// TwinCAT 3 PLC project LEO_Demo
// ProgramVersion: 3.1.4023.0
// libraries:
//   EfficientIO Communicator, * (EfficientIO)
//   Tc2_BABasic, * (Beckhoff Automation GmbH)
//   Tc2_Standard, * (Beckhoff Automation GmbH)
//   Tc2_System, * (Beckhoff Automation GmbH)
//   Tc2_Utilities, * (Beckhoff Automation GmbH)
//   Tc3_Module, * (Beckhoff Automation GmbH)
// project tree:
//   / FastTask.TcTTO, PlcTask.TcTTO, SlowTask.TcTTO
//   GVLs/ GVL.TcGVL
//   POUs/ prgComLynus.TcPOU, prgCS.TcPOU, prgEM.TcPOU, prgGrid.TcPOU, prgLightSwitch.TcPOU, prgPV.TcPOU, prgReadWrite.TcPOU, prgSun.TcPOU, prgSystemTime.TcPOU, prgVarInfo.TcPOU
// real-time tasks:
//   TASK MiddleTask: cycle T#10ms, priority 8, ADS port 350
//   TASK SlowTask: cycle T#20ms, priority 10, ADS port 351
//   TASK FastTask: cycle T#5ms, priority 6, ADS port 352

CONFIGURATION LEO_Demo
    RESOURCE PLC ON TwinCAT3
        TASK FastTask(INTERVAL := T#5ms, PRIORITY := 6);
        TASK PlcTask(INTERVAL := T#10ms, PRIORITY := 8);
        TASK SlowTask(INTERVAL := T#20ms, PRIORITY := 10);
        PROGRAM prgVarInfo WITH FastTask : prgVarInfo;
        PROGRAM prgReadWrite WITH FastTask : prgReadWrite;
        PROGRAM prgEM WITH PlcTask : prgEM;
        PROGRAM prgLightSwitch WITH PlcTask : prgLightSwitch;
        PROGRAM prgCS WITH PlcTask : prgCS;
        PROGRAM prgPV WITH PlcTask : prgPV;
        PROGRAM prgGrid WITH PlcTask : prgGrid;
        PROGRAM prgSystemTime WITH PlcTask : prgSystemTime;
        PROGRAM prgSun WITH PlcTask : prgSun;
        PROGRAM prgComLynus WITH SlowTask : prgComLynus;
    END_RESOURCE
END_CONFIGURATION

// ---- GVLs/GVL.TcGVL
{attribute 'qualified_only'}
VAR_GLOBAL
	location_lat	: LREAL; //{#lynus.ag#()}
	location_lon	: LREAL; //{#lynus.ag#()}
END_VAR

// ---- POUs/prgVarInfo.TcPOU
PROGRAM prgVarInfo
VAR
	fbVar			: FB_VarInfo;
END_VAR

fbVar(
	bReadInfo:= , 
	eTMCFile:= eSelectTMCFile.eDontUseTMCFile, 
	eSavePositionTMCFile:= eSavePositionOnPLC.ePostionC, 
	udiCounterFoundVariables=> , 
	bError=> , 
	bBusy=> , 
	byProgress=> , 
	udiErrorCodeOut=> , 
	eErrorVarInfo_Out=> , 
	sVarWithError=> );

END_PROGRAM

// ---- POUs/prgReadWrite.TcPOU
PROGRAM prgReadWrite
VAR
	fbRW		: FB_ReadWrite;
END_VAR

fbRW(bBusy=> , bError=> , udiErrorCodeOut=> , eErrorReadWrite_Out=> );

END_PROGRAM

// ---- POUs/prgEM.TcPOU
PROGRAM prgEM
VAR
	fbRand			: DRAND;
	lrRandNum		: LREAL;
	lrEMConsumption	: LREAL; //{#lynus.ag#()}
	lrEMCounter		: LREAL; //{#lynus.ag#()}
	fbTimer1		: TON;
	bStart1			: BOOL := TRUE;
	fbTimer2		: TON;
	bStart2			: BOOL;
END_VAR

fbTimer1(IN := bStart1, PT := T#15M);

IF fbTimer1.Q THEN
	bStart1 := FALSE;
	fbRand(Seed := 0);
	lrEMConsumption := fbRand.Num / 2;
	lrEMCounter := lrEMCounter + lrEMConsumption;
	bStart2 := TRUE;
END_IF

fbTimer2(IN := bStart2, PT := T#15M);

IF fbTimer2.Q THEN
	bStart2 := FALSE;
	fbRand(Seed := 0);
	lrEMConsumption := fbRand.Num;
	bStart1 := TRUE;
	lrEMCounter := lrEMCounter + lrEMConsumption;
END_IF

END_PROGRAM

// ---- POUs/prgLightSwitch.TcPOU
PROGRAM prgLightSwitch
VAR
	fbLight : FB_Light;
	bSwitchOn : BOOL; //{#lynus.ag#()}
	bSwitchOff : BOOL; //{#lynus.ag#()}
	bStateLight : BOOL; //{#lynus.ag#()}
END_VAR

fbLight(bOn:=bSwitchOn, bOff:=bSwitchOff, bLight=>bStateLight);

END_PROGRAM

// ---- POUs/prgCS.TcPOU
PROGRAM prgCS
VAR
	fbCSvirt	: FB_Light;
	bCSOn		: BOOL; //{#lynus.ag#()}
	bCSOff		: BOOL; //{#lynus.ag#()}
	bStateCS	: BOOL; //{#lynus.ag#()}
	lrCSpower	: LREAL; //{#lynus.ag#()}
END_VAR

fbCSvirt(bOn:=bCSOn, bOff:=bCSOff, bLight=>bStateCS);

IF bStateCS THEN
	lrCSpower := 11.02;
	ELSE
	lrCSpower := 0;
END_IF

END_PROGRAM

// ---- POUs/prgPV.TcPOU
PROGRAM prgPV
VAR
	fbPVvirt	: FB_Light;
	bPVOn		: BOOL; //{#lynus.ag#()}
	bPVOff		: BOOL; //{#lynus.ag#()}
	bStatePV	: BOOL; //{#lynus.ag#()}
	lrPVpower	: LREAL; //{#lynus.ag#()}
END_VAR

fbPVvirt(bOn:=bPVOn, bOff:=bPVOff, bLight=>bStatePV);

IF bStatePV THEN
	lrPVpower := 9.72;
	ELSE
	lrPVpower := 0;
END_IF

END_PROGRAM

// ---- POUs/prgGrid.TcPOU
PROGRAM prgGrid
VAR
	lrGridPower	: LREAL; //{#lynus.ag#()}
END_VAR

lrGridPower := prgEM.lrEMConsumption + prgCS.lrCSpower - prgPV.lrPVpower;

END_PROGRAM

// ---- POUs/prgSystemTime.TcPOU
PROGRAM prgSystemTime
VAR
	fbGetTime			: NT_GetTime;
	dtSystemTime		: DT;
	stDateTime			: TIMESTRUCT;
	tonGetTime			: TON;
	nStep				: INT;
	bSystemTimeValid	: BOOL := FALSE;
END_VAR

CASE nStep OF
0:
	tonGetTime(IN:=TRUE, PT:=T#500MS);
	IF (tonGetTime.Q) THEN
		tonGetTime(IN := FALSE);
		nStep:=10;
	END_IF

10:
	fbGetTime(NETID:='', START:=TRUE, TMOUT:=T#2S);
	IF (NOT fbGetTime.BUSY) THEN
		stDateTime := fbGetTime.TIMESTR;
		dtSystemTime := SYSTEMtimE_TO_DT(fbGetTime.TIMESTR);
		fbGetTime(START := FALSE);
		bSystemTimeValid := TRUE;
		nStep := 0;
	END_IF	
END_CASE

END_PROGRAM

// ---- POUs/prgSun.TcPOU
PROGRAM prgSun
VAR
	fbTimerC1					: FB_WeeklyTimeSwitch;
	fbCalcSunriseSunset   		: FB_CalcSunriseSunset;
	todSunrise            		: TOD;
	todSunset             		: TOD;
	bCircle1On					: BOOL;
	bCircle1Off					: BOOL;
	tSwitchOnTime				: TOD;	//{#lynus.ag#()}
	tSwitchOffTime				: TOD;	//{#lynus.ag#()}
END_VAR

VAR PERSISTENT
	bEnableTimerC1				: BOOL;
END_VAR


IF prgSystemTime.bSystemTimeValid THEN

	fbCalcSunriseSunset(
		fDegreeOfLongitude := GVL.location_lon,   (* Longitude of Verl *)
        fDegreeOfLatitude := GVL.location_lat,   (* Latitude of Verl *)
    	fReferenceMeridian := 30.0,  (* Central European Summer Time *)
        dCurrentDate := DT_TO_DATE(prgSystemTime.dtSystemTime),
        todSunrise => todSunrise,
        todSunset => todSunset);
END_IF


(*
IF prgSystemTime.bSystemTimeValid THEN

	fbTimerC1(
		bEnable:=bEnableTimerC1, 
		tCurrentDateTime:=prgSystemTime.dtSystemTime, 
		tSwitchOnTime:=todSunrise, 
		tSwitchOffTime:=todSunset, 
		bSunday:=TRUE, 
		bMonday:=TRUE, 
		bTuesday:=TRUE, 
		bWednesday:=TRUE, 
		bThursday:=TRUE, 
		bFriday:=TRUE, 
		bSaturday:=TRUE,
		bEdgeOn=> bCircle1On,
		bEdgeOff=> bCircle1Off);
END_IF
*)

END_PROGRAM

// ---- POUs/prgComLynus.TcPOU
PROGRAM prgComLynus
VAR
	fbCom			: FB_MqttCommunicator;
END_VAR

fbCom(
	bConnect:= TRUE, 
	sUserName:= 'c43048fc-b368-4152-a20e-2efdedf6f25a', 
	sUserPassword:= 'a3dbe556-ed89-450d-a0be-4c95c1f665ec', 
	eSavePositionCertificate:= eSavePositionOnPLC.ePostionC, 
	bConnected=> , 
	bError=> , 
	hrErrorCode=> , 
	eConnectionState=> , 
	eErrorMessage_Out=> );

END_PROGRAM
